{attribute 'linkalways'} 
{attribute 'no_explicit_call' := 'This FB is a CLASS and must be accessed using methods or properties'}
{attribute 'enable_dynamic_creation'}
FUNCTION_BLOCK Node_F_VN_ConvexityDefects EXTENDS VisionNode
VAR
    ipContour : _ITcVnContainer;
    ipConvexityDefects : _ITcVnContainer;
    hrPrev : _HRESULT(S_OK);
	hresult : _HRESULT(S_OK);
END_VAR

METHOD PUBLIC  Clone : I_Node
VAR
	pNode : POINTER TO Node_F_VN_ConvexityDefects;
END_VAR
pNode := __NEW(Node_F_VN_ConvexityDefects);
Clone := pNode^;
END_METHOD

METHOD FB_init : BOOL
VAR_INPUT
	bInitRetains : BOOL; // if TRUE, the retain variables are initialized (warm start / cold start)
	bInCopyCode : BOOL;  // if TRUE, the instance afterwards gets moved into the copy code (online change)
END_VAR
AddInput('ipContour', ipContour);
AddInput('hrPrev', hrPrev);
AddOutput('ipConvexityDefects', ipConvexityDefects);
AddOutput('hresult',hresult);
END_METHOD

METHOD PROTECTED OnExecute
hresult.Value := F_VN_ConvexityDefects(
	ipContour := ipContour.Value,
    ipConvexityDefects := ipConvexityDefects.Value,
	hrPrev:= hrPrev.Value);
END_METHOD

METHOD PUBLIC PreExecutionCheck
VAR_INPUT
	Check : I_PreExecutionChecks;
END_VAR
Check.IsTrue(ipContour.IsValid, 'ipContour must be a valid container');
Check.IsTrue(ipContour.IsType(TC_GLOBAL_CONST_LIST.ContainerType_Vector_TcVnPoint2_DINT), 'ipContour contains incorrect type');
END_METHOD

END_FUNCTION_BLOCK

(* stored: Version 1.1.0.1, ProductVersion 3.1.4026.13
   POU Node_F_VN_ConvexityDefects: Id {a3f1faa1-f766-0867-0ef5-b27dc52c47e7}, SpecialFunc None
   Folder Constructor: Id {24c672dd-08ae-004d-0e05-f0e0fa83ed77}
   Method Clone: Id {ccf7944d-7b2c-0b9d-0a49-8830ff5fb484}
   Method FB_init: Id {5792a211-45ac-0f83-2cb1-223b2c57cef7}
   Method OnExecute: Id {e9d30748-7a1c-084b-008b-61fdc6c9195a}
   Method PreExecutionCheck: Id {a00b80b2-ecf3-056c-16de-edafe02f341e} *)
